// Mitsubishi GX Works2 project: z06   PLC: Q02/Q02H

PROGRAM MAIN
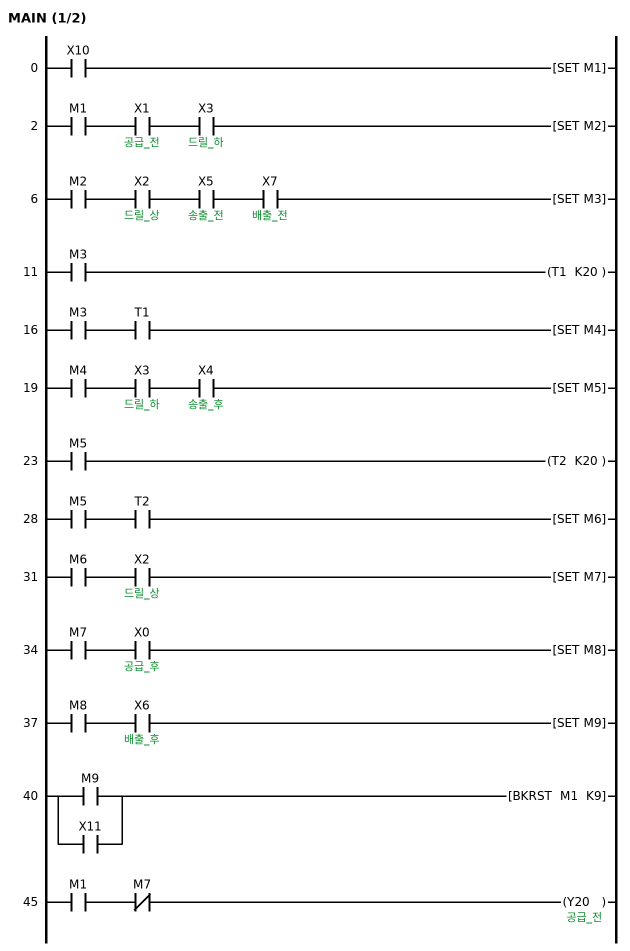
0     LD      X10
      SET     M1
2     LD      M1
      AND     X1  ; 공급_전
      AND     X3  ; 드릴_하
      SET     M2
6     LD      M2
      AND     X2  ; 드릴_상
      AND     X5  ; 송출_전
      AND     X7  ; 배출_전
      SET     M3
11    LD      M3
      OUT     T1 K20
16    LD      M3
      AND     T1
      SET     M4
19    LD      M4
      AND     X3  ; 드릴_하
      AND     X4  ; 송출_후
      SET     M5
23    LD      M5
      OUT     T2 K20
28    LD      M5
      AND     T2
      SET     M6
31    LD      M6
      AND     X2  ; 드릴_상
      SET     M7
34    LD      M7
      AND     X0  ; 공급_후
      SET     M8
37    LD      M8
      AND     X6  ; 배출_후
      SET     M9
40    LD      M9
      OR      X11
      BKRST   M1 K9
45    LD      M1
      ANI     M7
      OUT     Y20  ; 공급_전
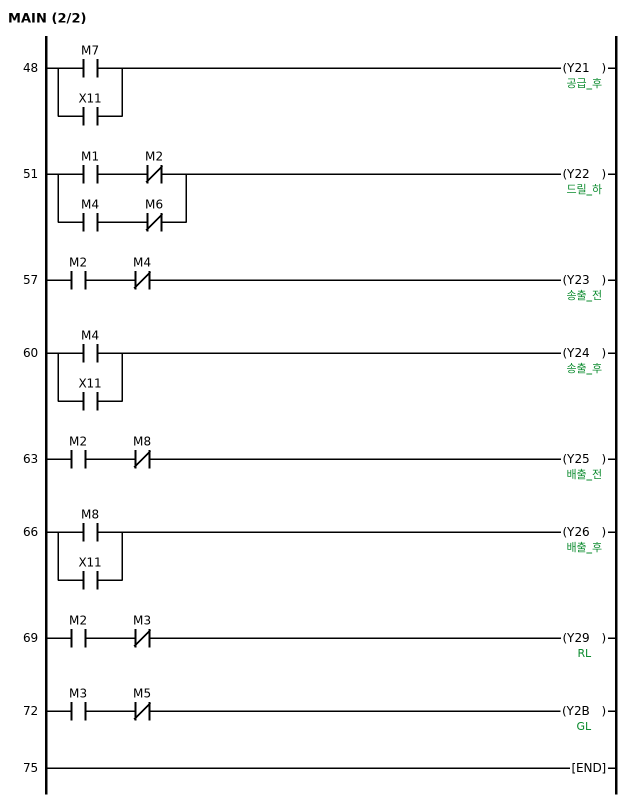
48    LD      M7
      OR      X11
      OUT     Y21  ; 공급_후
51    LD      M1
      ANI     M2
      LD      M4
      ANI     M6
      ORB
      OUT     Y22  ; 드릴_하
57    LD      M2
      ANI     M4
      OUT     Y23  ; 송출_전
60    LD      M4
      OR      X11
      OUT     Y24  ; 송출_후
63    LD      M2
      ANI     M8
      OUT     Y25  ; 배출_전
66    LD      M8
      OR      X11
      OUT     Y26  ; 배출_후
69    LD      M2
      ANI     M3
      OUT     Y29  ; RL
72    LD      M3
      ANI     M5
      OUT     Y2B  ; GL
75    END
END_PROGRAM

// device comments not shown above
Y2A  ; YL
